FUNCTION FC_StringNotEmpty : BOOL
VAR_INPUT
	iString:	T_DEFAULT_STR;
END_VAR

FC_StringNotEmpty := LEN(iString) > 0;

END_FUNCTION

(* stored: Version 1.1.0.1, ProductVersion 3.1.4026.18
   POU FC_StringNotEmpty: Id {0894167f-e28b-4e0b-a863-a5145ce50d2e}, SpecialFunc None *)
